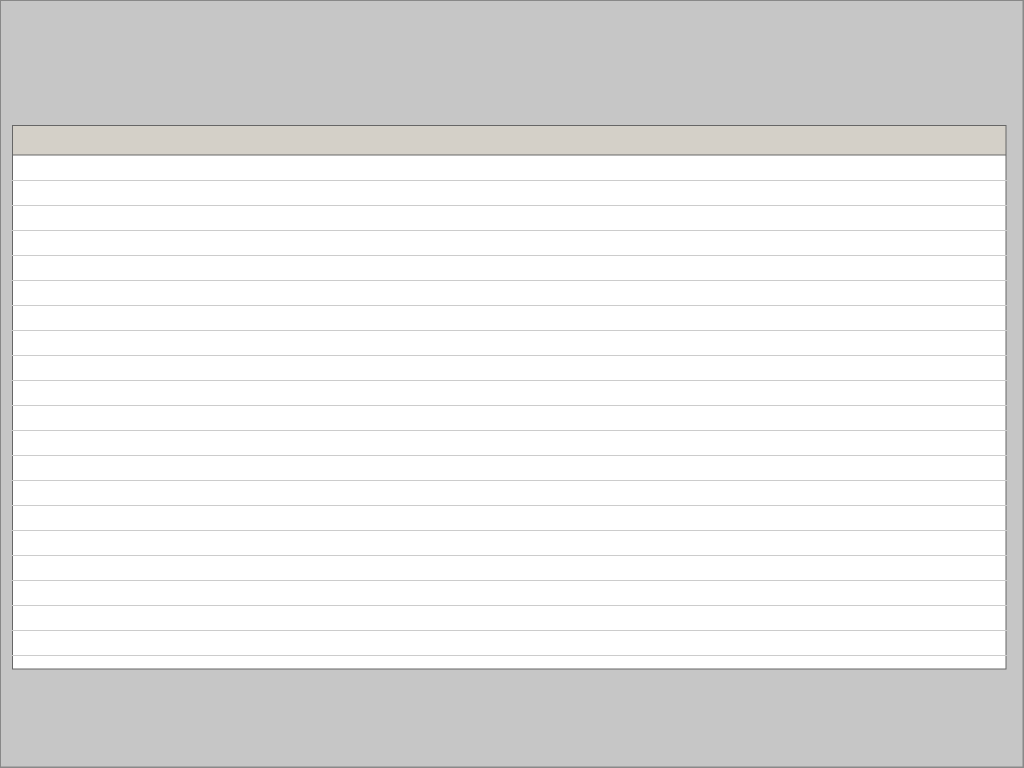
VISUALIZATION SS_12_AlarmsTest  // 1024x768
    Frame (0,0 1024x768)
        shows SS_91_Template(header := HMIData.hmiHeader)
    Table (12,125 994x544), data array: msgTest.msgArry
        p3854506369: msgTest.msgArry[INDEX].timeRaised
        p1892666644: msgTest.msgArry[INDEX].timeResolved
        p338671338: msgTest.msgArry[INDEX].text
        p2170511999: msgTest.msgArry[INDEX].source
        p2232123230: Time Raised
        p511219082: Time Resolved
        p1755163831: Message Text
        p4092479075: Fault Location
        Columns.Column.[0].Template: msgTest.msgArryStyle[INDEX].isColoured; msgTest.msgArryStyle[INDEX].colourToApply
        Columns.Column.[1].Template: msgTest.msgArryStyle[INDEX].isColoured; msgTest.msgArryStyle[INDEX].colourToApply
        Columns.Column.[2].Template: msgTest.msgArryStyle[INDEX].isColoured; msgTest.msgArryStyle[INDEX].colourToApply
        Columns.Column.[3].Template: msgTest.msgArryStyle[INDEX].isColoured; msgTest.msgArryStyle[INDEX].colourToApply
END_VISUALIZATION

(* stored: Version 1.1.0.1, ProductVersion 3.1.4024.12
   Visu SS_12_AlarmsTest: Id {f0caa955-e950-4402-b6fa-6d4c00190f55} *)
